PROGRAM MAIN
VAR
	fbWave			: FB_SquareWave;
	fbToggle		: FB_ToggleSwitch;
	
	fbInletConv		: FB_Conveyor;
	fbConveyor		: FB_Conveyor;
	fbConveyor_2	: FB_Conveyor;
	fbConveyor_3	: FB_Conveyor;
	
	fbActuator		: FB_Actuator;
	
	iPulseLength	: DINT;
	
	testInt			: REAL;
	sequenceStep	: INT;
	
	handover		: BOOL;
	
	GoToWork		: BOOL;
	GoToHome		: BOOL;
	InWork			: BOOL;
	InHome			: BOOL;
	
END_VAR


iPulseLength := DataExchange.iVar1;	// helper variable - pulse length in ms

fbWave(PulseLength := iPulseLength);	// instance of FB_SquareWave

DataExchange.bVar1 := fbWave.Value;

fbToggle(
	switch := DataExchange.button1,
	status => DataExchange.status1);

fbActuator(
	Sensor_Work := DataExchange.DAC_Sens_Work,
	Sensor_Home := DataExchange.DAC_Sens_Home,
	GoToPos_Work := GoToWork,
	GoToPos_Home := GoToHome,
	ToPos_Work => DataExchange.DAC_Coil_Work,
	ToPos_Home => DataExchange.DAC_Coil_Home,
	InPos_Work => InWork,
	InPos_Home => InHome);
	
fbInletConv(
	Occupied := 	DataExchange.sensor1,
	Handover := 	handover AND fbConveyor.Taking,
	Takeover :=		fbConveyor_3.Giving OR sequenceStep = 10,
	EnableMotor =>	DataExchange.motor1
);
	
fbConveyor(
	Occupied := 	DataExchange.sensor2,
	Handover := 	fbConveyor_2.Taking,
	Takeover :=		fbInletConv.Giving,
	EnableMotor =>	DataExchange.motor2
);

fbConveyor_2(
	Occupied := 	DataExchange.sensor3,
	Handover := 	fbConveyor_3.Taking,
	Takeover :=		fbConveyor.Giving,
	EnableMotor =>	DataExchange.motor3
);

fbConveyor_3(
	Occupied := 	DataExchange.sensor4,
	Handover := 	fbInletConv.Taking,
	Takeover :=		fbConveyor_2.Giving,
	EnableMotor =>	DataExchange.motor4
);



CASE sequenceStep OF
	0: 
		handover := FALSE;
		IF DataExchange.pusherRetracted OR NOT DataExchange.pusherExtended THEN
			IF DataExchange.retracted OR NOT DataExchange.extended THEN
				DataExchange.extend := TRUE;
				DataExchange.retract := FALSE;				
			END_IF
		ELSE
			DataExchange.pusherBwd := TRUE;
			DataExchange.pusherFwd := FALSE;
		END_IF
		
		IF (DataExchange.pusherRetracted OR NOT DataExchange.pusherExtended) AND DataExchange.extended THEN
			sequenceStep := 10;
		END_IF
	10:
		IF DataExchange.sensor1 AND NOT DataExchange.motor1 THEN
			DataExchange.pusherFwd := TRUE;
			DataExchange.pusherBwd := FALSE;
		END_IF	
		IF DataExchange.pusherExtended THEN
			sequenceStep := 20;
		END_IF
	20: 
		DataExchange.pusherBwd := TRUE;
		DataExchange.pusherFwd := FALSE;
		IF DataExchange.pusherRetracted THEN
			sequenceStep := 30;
		END_IF
	30: 
		DataExchange.extend := FALSE;
		DataExchange.retract := TRUE;	
		IF DataExchange.retracted THEN
			handover := TRUE;
			sequenceStep := 40;
		END_IF
	40: 
		IF NOT DataExchange.sensor1 THEN
			handover := FALSE;
			sequenceStep := 0;
		END_IF
END_CASE

END_PROGRAM

(* stored: Version 1.1.0.1, ProductVersion 3.1.4022.18
   POU MAIN: Id {9ab6868b-4f3c-4c35-b59f-5ea0a58ab847}, SpecialFunc None *)
